PROGRAM MAIN
VAR
	bTestSimple: BOOL;
END_VAR

END_PROGRAM

(* stored: Version 1.1.0.1, ProductVersion 3.1.4024.16
   POU MAIN: Id {23b953e1-d7ce-4d73-a12b-a9dba7f63728}, SpecialFunc None *)
